// Mitsubishi GX Works2 project: servo_motor_intro   PLC: Q02/Q02H

PROGRAM MAIN
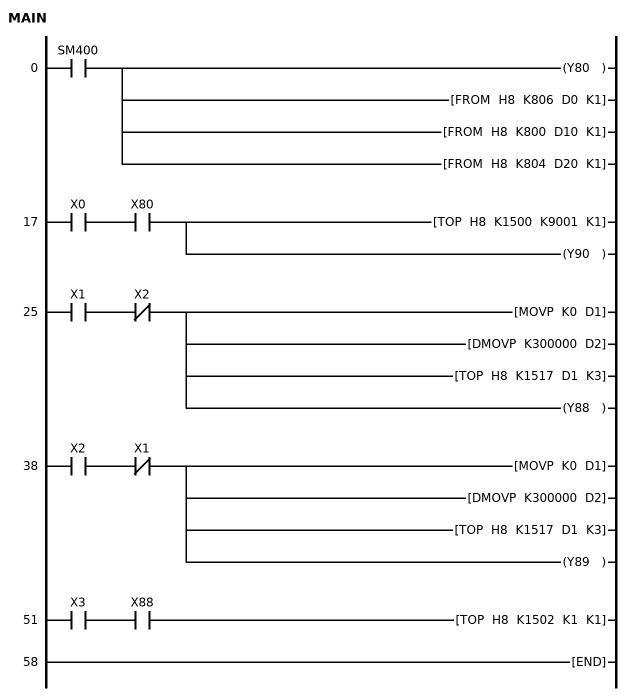
0     LD      SM400
      OUT     Y80
      FROM    H8 K806 D0 K1
      FROM    H8 K800 D10 K1
      FROM    H8 K804 D20 K1
17    LD      X0
      AND     X80
      TOP     H8 K1500 K9001 K1
      OUT     Y90
25    LD      X1
      ANI     X2
      MOVP    K0 D1
      DMOVP   K300000 D2
      TOP     H8 K1517 D1 K3
      OUT     Y88
38    LD      X2
      ANI     X1
      MOVP    K0 D1
      DMOVP   K300000 D2
      TOP     H8 K1517 D1 K3
      OUT     Y89
51    LD      X3
      AND     X88
      TOP     H8 K1502 K1 K1
58    END
END_PROGRAM
